{attribute 'GeneratedUsingTerminal: KL6904'}
{attribute addProperty BoxType "KL6904"}
{attribute addProperty Id "Channel_1AT %Q*Channel_9E2936860"}
{attribute addProperty CRC "3107509778"}
{attribute addProperty Size "0"}
TYPE KL6904_B938D612 :
STRUCT
	{attribute addProperty Name "Channel_1"}
	Channel_1 : Channel_9E293686;
END_STRUCT
END_TYPE

(* stored: Version 1.2.0.0, ProductVersion 3.1.4024.9
   DUT KL6904_B938D612: Id {7267c065-d753-453b-b01e-e904000ad600} *)
